{region '#Template'}
	{attribute 'Version' := '1.2.0.0'}
	{attribute 'Tags' := '"LCID": "1031", "Text": "Types, Publisher, Subscriber, Weather, Data"'}
	{attribute 'Tags' := '"LCID": "1033", "Text": "Types, Publisher, Subscriber, Weather, Data"'}
	{attribute 'Description' := '"LCID": "1031", "Text": "Daten Wetterstation"'}
	{attribute 'Description' := '"LCID": "1033", "Text": "Weatherstation-data"'}
{endregion}
TYPE ST_BA_WeatherStation :
STRUCT
	bDisturb				: BOOL;
	fLatitude				: REAL;				// [°]
	fLongitude				: REAL;				// [°]
	fSunAzimuth				: REAL;				// [°]
	fSunElevation			: REAL;				// [°]
	bRain					: BOOL;
	stDateTime				: TIMESTRUCT;
	fOutsideTemperature		: REAL;				// [°C]
	fDewPointTemperature	: REAL;				// [°C]		 
	fPressureAbs			: REAL;				// [hPa]
	fPressureRel			: REAL;				// [hPa]			 
	fHumidityAbs			: REAL;				// [g/m³]
	fHumidityRel			: REAL;				// [%rF]	
	fBrightnessNorth		: REAL;				// [Lux]		 
	fBrightnessEast			: REAL;				// [Lux]
	fBrightnessSouth		: REAL;				// [Lux]
	fBrightnessWest			: REAL;				// [Lux]			 
	fDawn					: REAL;				// [Lux] 
	fGlobalRadiation		: REAL;				// [W/m²]			 
	fWindDirection			: REAL;				// [°]
	fWindSpeed				: REAL;				// [m/s]
END_STRUCT
END_TYPE

(* stored: Version 1.1.0.1, ProductVersion 3.1.4024.9
   DUT ST_BA_WeatherStation: Id {c78e9017-6f4b-4c0c-aa38-a73a8938c63a} *)
